(* IEC 61131-3 sources: repolevel_ST_code_completion/real_groud_truth最新/repoeval_PID_controller/readful_result, 2 files *)

(* ---- PID_controller.st ---- *)
//***************************************************************
//* Continue defining the internal variables and logic for the PID controller
//***************************************************************
VAR
    err: REAL; // Error (SP - PV)
    prev_err: REAL := 0; // Previous error
    integral: REAL := 0; // Integral accumulator
    derivative: REAL := 0; // Derivative term
    prev_PV: REAL := 0; // Previous process variable
    last_time: TIME := T#0ms; // Last execution time
END_VAR

//***************************************************************
//* Initialization logic
//***************************************************************
IF last_time = T#0ms THEN
    last_time := TIME(); // Initialize the last execution time
END_IF

//***************************************************************
//* Main PID calculation logic
//***************************************************************
err := SP - PV; // Calculate error

// Proportional term
CO_P := Kc * err;

// Integral term
integral := integral + (err * TO_REAL(SampleTime) / TO_REAL(millis));
CO_I := Kc * (integral / Ti);

// Derivative term
IF SampleTime > T#0ms THEN
    derivative := (PV - prev_PV) / TO_REAL(SampleTime);
END_IF
CO_D := -Kc * Td * derivative;

// Calculate the total controller output
CO := CO_P + CO_I + CO_D;

// Apply output limits
IF CO > UpperLimit THEN
    CO := UpperLimit;
ELSIF CO < LowerLimit THEN
    CO := LowerLimit;
END_IF

// Update previous values for the next iteration
prev_err := err;
prev_PV := PV;
last_time := TIME();

(* ---- Tank.st ---- *)
// Internal variables for simulation
VAR
    DeltaTime: REAL; // Time step in seconds
    FlowChange: REAL; // Change in tank level based on input/output flow
END_VAR

// Calculate the time step in seconds
DeltaTime := REAL_TO_TIME(SampleTime) / T#1s;

// Calculate the change in tank level based on input and output flow
FlowChange := (Process_In - Process_Out) * DeltaTime;

// Update the tank level
Level := Level + FlowChange;

// Ensure the tank level stays within the defined limits
IF Level < Lower_limit THEN
    Level := Lower_limit;
ELSIF Level > Upper_limit THEN
    Level := Upper_limit;
END_IF;
END_FUNCTION_BLOCK
